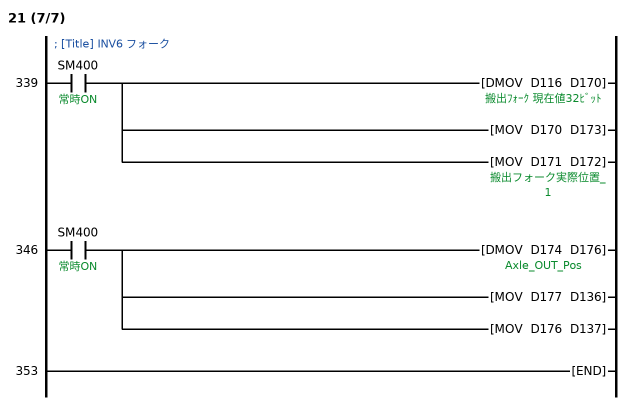
; [Title] INV6 フォーク
339   LD      SM400  ; 常時ON
      DMOV    D116 D170  ; 搬出ﾌｫｰｸ 現在値32ﾋﾞｯﾄ
      MOV     D170 D173
      MOV     D171 D172
346   LD      SM400  ; 常時ON
      DMOV    D174 D176
      MOV     D177 D136
      MOV     D176 D137
353   END
END_PROGRAM

PROGRAM 22  // Drive
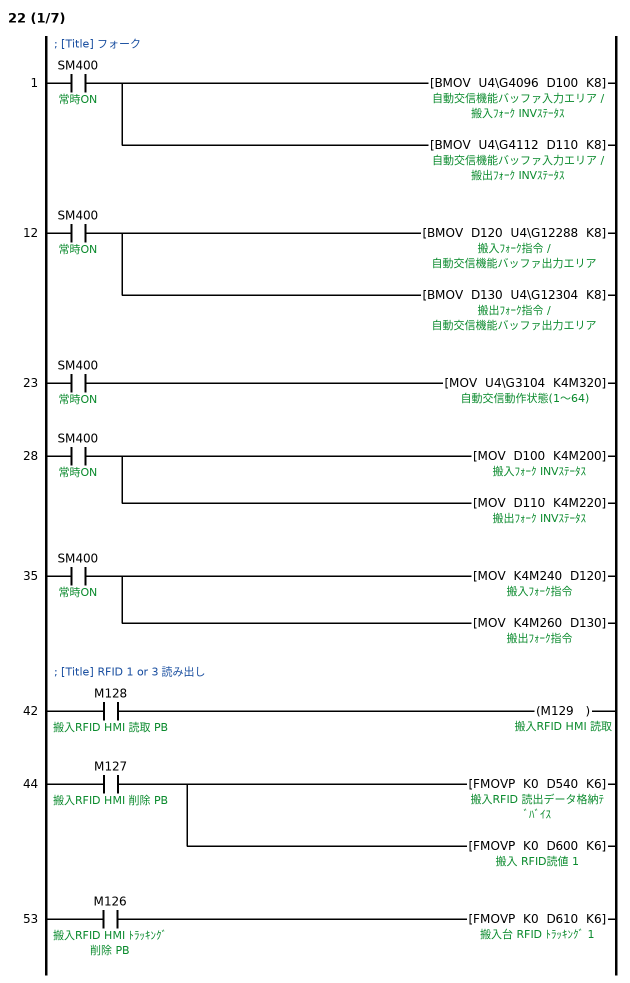
; [Title] フォーク
1     LD      SM400  ; 常時ON
      BMOV    U4\G4096 D100 K8  ; 自動交信機能バッファ入力エリア / 搬入ﾌｫｰｸ INVｽﾃｰﾀｽ
      BMOV    U4\G4112 D110 K8  ; 自動交信機能バッファ入力エリア / 搬出ﾌｫｰｸ INVｽﾃｰﾀｽ
12    LD      SM400  ; 常時ON
      BMOV    D120 U4\G12288 K8  ; 搬入ﾌｫｰｸ指令 / 自動交信機能バッファ出力エリア
      BMOV    D130 U4\G12304 K8  ; 搬出ﾌｫｰｸ指令 / 自動交信機能バッファ出力エリア
23    LD      SM400  ; 常時ON
      MOV     U4\G3104 K4M320  ; 自動交信動作状態(1～64) / INV2 通信異常
28    LD      SM400  ; 常時ON
      MOV     D100 K4M200  ; 搬入ﾌｫｰｸｽﾃｰﾀｽ 未使用
      MOV     D110 K4M220  ; 搬出ﾌｫｰｸｽﾃｰﾀｽ 未使用
35    LD      SM400  ; 常時ON
      MOV     K4M240 D120  ; 搬入ﾌｫｰｸ緊急停止
      MOV     K4M260 D130  ; 搬出ﾌｫｰｸ緊急停止
; [Title] RFID 1 or 3 読み出し
42    LD      M128  ; 搬入RFID HMI 読取 PB
      OUT     M129  ; 搬入RFID HMI 読取
44    LD      M127  ; 搬入RFID HMI 削除 PB
      FMOVP   K0 D540 K6  ; 搬入RFID 読出データ格納ﾃﾞﾊﾞｲｽ
      FMOVP   K0 D600 K6  ; 搬入 RFID読値 1
53    LD      M126  ; 搬入RFID HMI ﾄﾗｯｷﾝｸﾞ 削除 PB
      FMOVP   K0 D610 K6  ; 搬入台 RFID ﾄﾗｯｷﾝｸﾞ 1
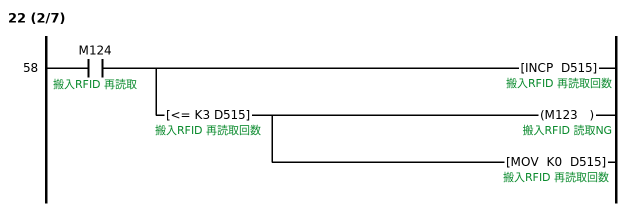
58    LD      M124  ; 搬入RFID 再読取
      INCP    D515  ; 搬入RFID 再読取回数
      AND<=   K3 D515  ; 搬入RFID 再読取回数
      OUT     M123  ; 搬入RFID 読取NG
      MOV     K0 D515
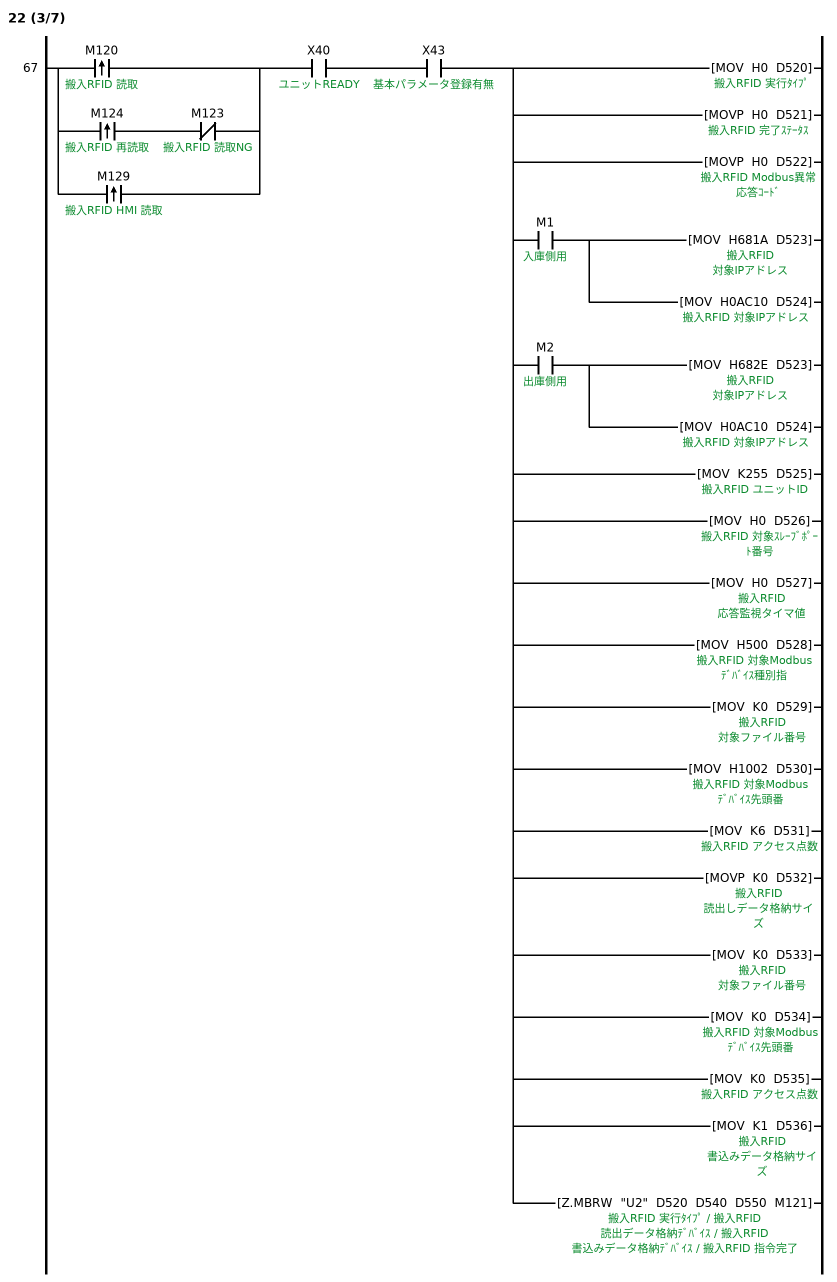
67    LDP     M120  ; 搬入RFID 読取
      LDP     M124  ; 搬入RFID 再読取
      ANI     M123  ; 搬入RFID 読取NG
      ORB
      ORP     M129  ; 搬入RFID HMI 読取
      AND     X40  ; ユニットREADY
      AND     X43  ; 基本パラメータ登録有無
      MOV     H0 D520  ; 搬入RFID 実行ﾀｲﾌﾟ
      MOVP    H0 D521  ; 搬入RFID 完了ｽﾃｰﾀｽ
      MOVP    H0 D522  ; 搬入RFID Modbus異常応答ｺｰﾄﾞ
      MPS
      AND     M1  ; 入庫側用
      MOV     H681A D523  ; 搬入RFID 対象IPアドレス
      MOV     H0AC10 D524  ; 搬入RFID 対象IPアドレス
      MRD
      AND     M2  ; 出庫側用
      MOV     H682E D523
      MOV     H0AC10 D524
      MPP
      MOV     K255 D525  ; 搬入RFID ユニットID
      MOV     H0 D526  ; 搬入RFID 対象ｽﾚｰﾌﾞﾎﾟｰﾄ番号
      MOV     H0 D527  ; 搬入RFID 応答監視タイマ値
      MOV     H500 D528  ; 搬入RFID 対象Modbusﾃﾞﾊﾞｲｽ種別指
      MOV     K0 D529  ; 搬入RFID 対象ファイル番号
      MOV     H1002 D530  ; 搬入RFID 対象Modbus ﾃﾞﾊﾞｲｽ先頭番
      MOV     K6 D531  ; 搬入RFID アクセス点数
      MOVP    K0 D532  ; 搬入RFID 読出しデータ格納サイズ
      MOV     K0 D533  ; 搬入RFID 対象ファイル番号
      MOV     K0 D534  ; 搬入RFID 対象Modbus ﾃﾞﾊﾞｲｽ先頭番
      MOV     K0 D535  ; 搬入RFID アクセス点数
      MOV     K1 D536  ; 搬入RFID 書込みデータ格納サイズ
      Z.MBRW  "U2" D520 D540 D550 M121  ; 搬入RFID 書込みデータ格納ﾃﾞﾊﾞｲｽ / 搬入RFID 指令完了
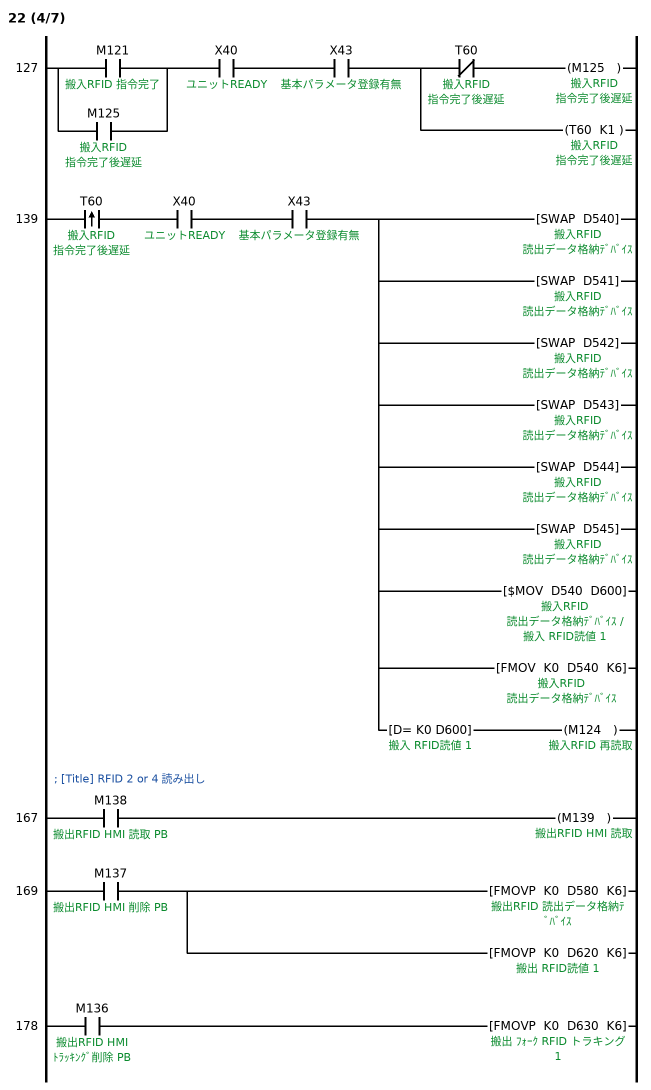
127   LD      M121  ; 搬入RFID 指令完了
      OR      M125  ; 搬入RFID 指令完了後遅延
      AND     X40  ; ユニットREADY
      AND     X43  ; 基本パラメータ登録有無
      MPS
      ANI     T60  ; 搬入RFID 指令完了後遅延
      OUT     M125  ; 搬入RFID 指令完了後遅延
      MPP
      OUT     T60 K1  ; 搬入RFID 指令完了後遅延
139   LDP     T60  ; 搬入RFID 指令完了後遅延
      AND     X40  ; ユニットREADY
      AND     X43  ; 基本パラメータ登録有無
      SWAP    D540
      SWAP    D541  ; 搬入RFID 読出データ格納ﾃﾞﾊﾞｲｽ
      SWAP    D542  ; 搬入RFID 読出データ格納ﾃﾞﾊﾞｲｽ
      SWAP    D543  ; 搬入RFID 読出データ格納ﾃﾞﾊﾞｲｽ
      SWAP    D544  ; 搬入RFID 読出データ格納ﾃﾞﾊﾞｲｽ
      SWAP    D545  ; 搬入RFID 読出データ格納ﾃﾞﾊﾞｲｽ
      $MOV    D540 D600
      FMOV    K0 D540 K6
      ANDD=   K0 D600  ; 搬入 RFID読値 1
      OUT     M124  ; 搬入RFID 再読取
; [Title] RFID 2 or 4 読み出し
167   LD      M138  ; 搬出RFID HMI 読取 PB
      OUT     M139  ; 搬出RFID HMI 読取
169   LD      M137  ; 搬出RFID HMI 削除 PB
      FMOVP   K0 D580 K6  ; 搬出RFID 読出データ格納ﾃﾞﾊﾞｲｽ
      FMOVP   K0 D620 K6  ; 搬出 RFID読値 1
178   LD      M136  ; 搬出RFID HMI ﾄﾗｯｷﾝｸﾞ削除 PB
      FMOVP   K0 D630 K6  ; 搬出 ﾌｫｰｸ RFID トラキング 1
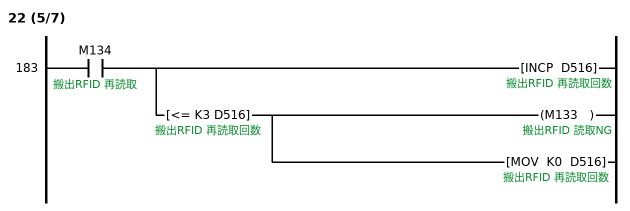
183   LD      M134  ; 搬出RFID 再読取
      INCP    D516  ; 搬出RFID 再読取回数
      AND<=   K3 D516  ; 搬出RFID 再読取回数
      OUT     M133  ; 搬出RFID 読取NG
      MOV     K0 D516
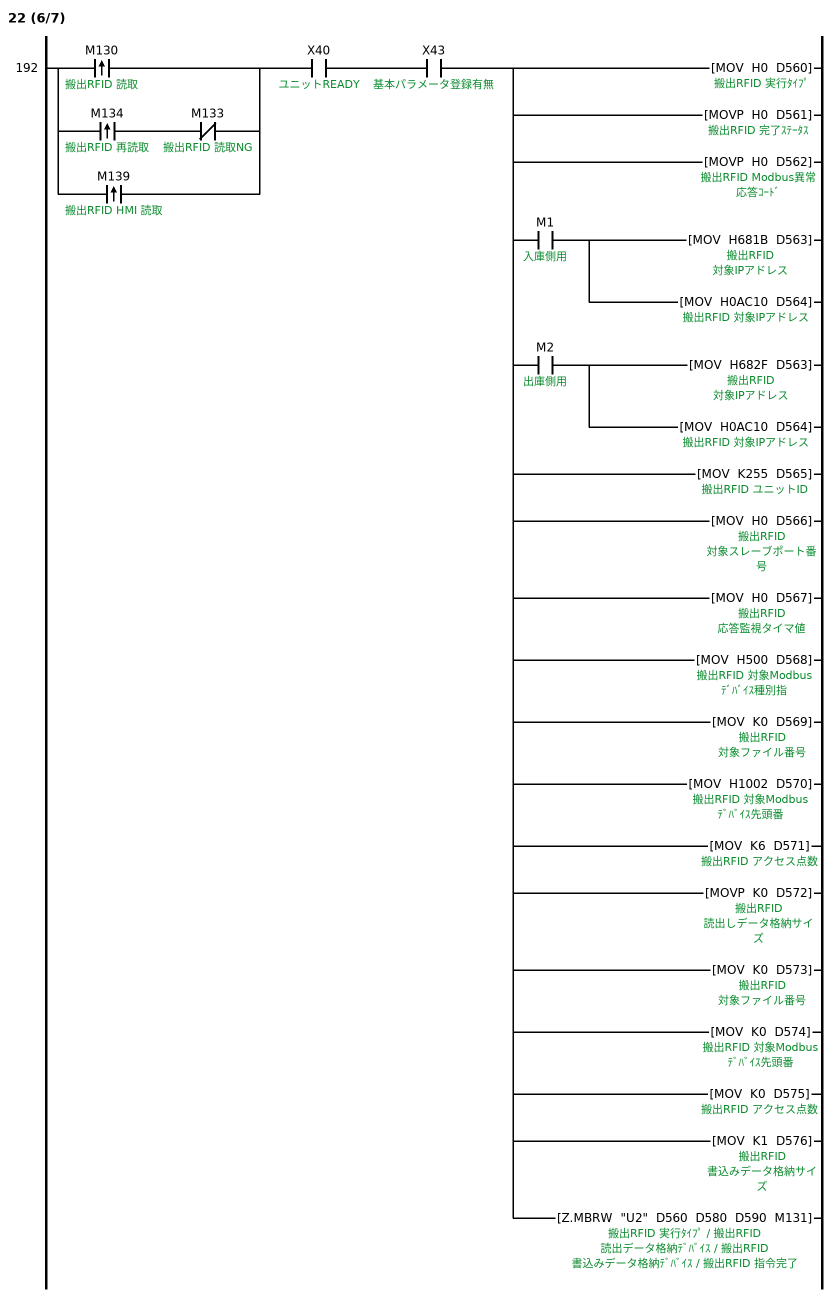
192   LDP     M130  ; 搬出RFID 読取
      LDP     M134  ; 搬出RFID 再読取
      ANI     M133  ; 搬出RFID 読取NG
      ORB
      ORP     M139  ; 搬出RFID HMI 読取
      AND     X40  ; ユニットREADY
      AND     X43  ; 基本パラメータ登録有無
      MOV     H0 D560  ; 搬出RFID 実行ﾀｲﾌﾟ
      MOVP    H0 D561  ; 搬出RFID 完了ｽﾃｰﾀｽ
      MOVP    H0 D562  ; 搬出RFID Modbus異常応答ｺｰﾄﾞ
      MPS
      AND     M1  ; 入庫側用
      MOV     H681B D563  ; 搬出RFID 対象IPアドレス
      MOV     H0AC10 D564  ; 搬出RFID 対象IPアドレス
      MRD
      AND     M2  ; 出庫側用
      MOV     H682F D563
      MOV     H0AC10 D564
      MPP
      MOV     K255 D565  ; 搬出RFID ユニットID
      MOV     H0 D566  ; 搬出RFID 対象スレーブポート番号
      MOV     H0 D567  ; 搬出RFID 応答監視タイマ値
      MOV     H500 D568  ; 搬出RFID 対象Modbusﾃﾞﾊﾞｲｽ種別指
      MOV     K0 D569  ; 搬出RFID 対象ファイル番号
      MOV     H1002 D570  ; 搬出RFID 対象Modbus ﾃﾞﾊﾞｲｽ先頭番
      MOV     K6 D571  ; 搬出RFID アクセス点数
      MOVP    K0 D572  ; 搬出RFID 読出しデータ格納サイズ
      MOV     K0 D573  ; 搬出RFID 対象ファイル番号
      MOV     K0 D574  ; 搬出RFID 対象Modbus ﾃﾞﾊﾞｲｽ先頭番
      MOV     K0 D575  ; 搬出RFID アクセス点数
      MOV     K1 D576  ; 搬出RFID 書込みデータ格納サイズ
      Z.MBRW  "U2" D560 D580 D590 M131  ; 搬出RFID 書込みデータ格納ﾃﾞﾊﾞｲｽ / 搬出RFID 指令完了
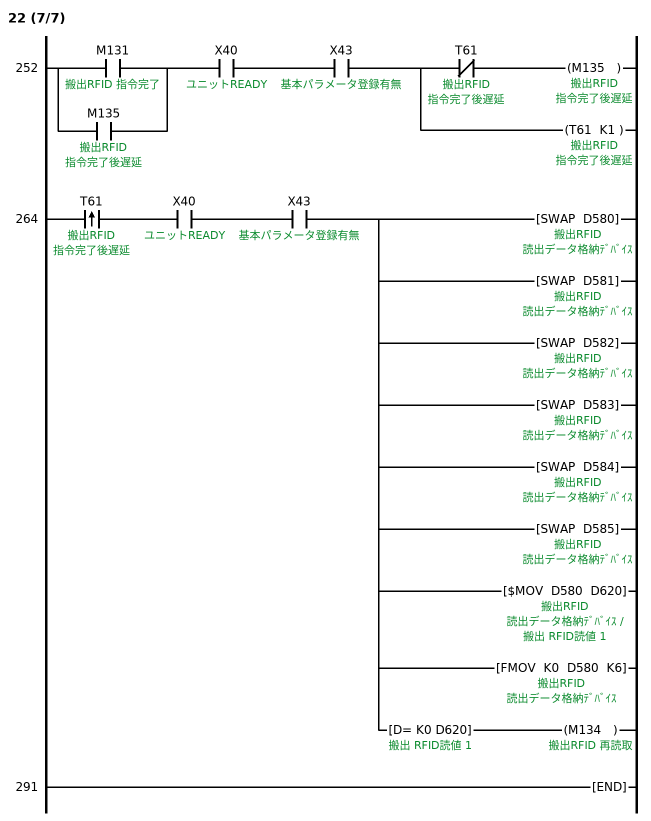
252   LD      M131  ; 搬出RFID 指令完了
      OR      M135  ; 搬出RFID 指令完了後遅延
      AND     X40  ; ユニットREADY
      AND     X43  ; 基本パラメータ登録有無
      MPS
      ANI     T61  ; 搬出RFID 指令完了後遅延
      OUT     M135  ; 搬出RFID 指令完了後遅延
      MPP
      OUT     T61 K1  ; 搬出RFID 指令完了後遅延
264   LDP     T61  ; 搬出RFID 指令完了後遅延
      AND     X40  ; ユニットREADY
      AND     X43  ; 基本パラメータ登録有無
      SWAP    D580
      SWAP    D581  ; 搬出RFID 読出データ格納ﾃﾞﾊﾞｲｽ
      SWAP    D582  ; 搬出RFID 読出データ格納ﾃﾞﾊﾞｲｽ
      SWAP    D583  ; 搬出RFID 読出データ格納ﾃﾞﾊﾞｲｽ
      SWAP    D584  ; 搬出RFID 読出データ格納ﾃﾞﾊﾞｲｽ
      SWAP    D585  ; 搬出RFID 読出データ格納ﾃﾞﾊﾞｲｽ
      $MOV    D580 D620
      FMOV    K0 D580 K6
      ANDD=   K0 D620  ; 搬出 RFID読値 1
      OUT     M134  ; 搬出RFID 再読取
291   END
END_PROGRAM

PROGRAM 30  // AGV
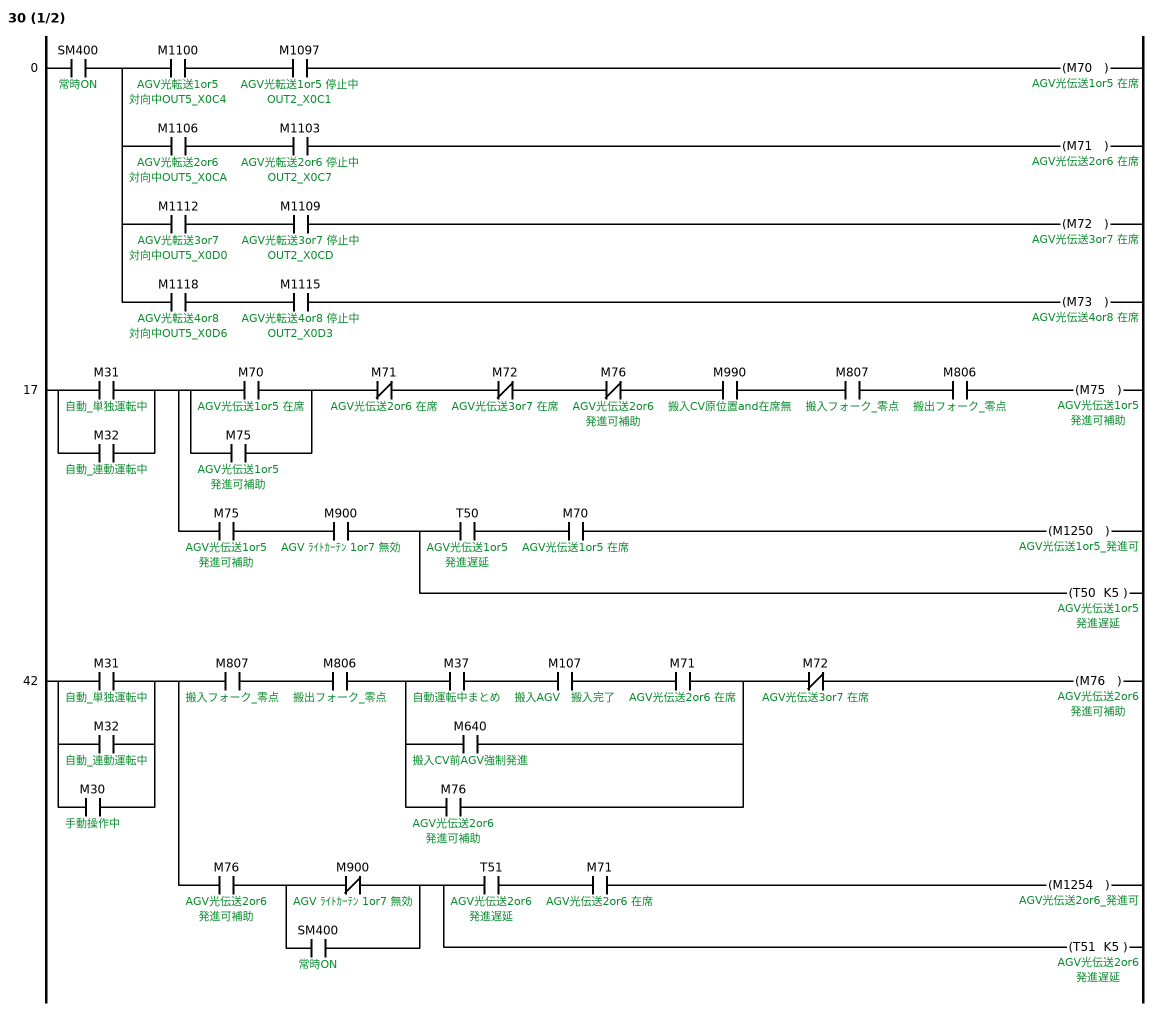
0     LD      SM400  ; 常時ON
      MPS
      AND     M1100  ; AGV光転送1or5 対向中OUT5_X0C4
      AND     M1097  ; AGV光転送1or5 停止中 OUT2_X0C1
      OUT     M70  ; AGV光伝送1or5 在席
      MRD
      AND     M1106  ; AGV光転送2or6 対向中OUT5_X0CA
      AND     M1103  ; AGV光転送2or6 停止中 OUT2_X0C7
      OUT     M71  ; AGV光伝送2or6 在席
      MRD
      AND     M1112  ; AGV光転送3or7 対向中OUT5_X0D0
      AND     M1109  ; AGV光転送3or7 停止中 OUT2_X0CD
      OUT     M72  ; AGV光伝送3or7 在席
      MPP
      AND     M1118  ; AGV光転送4or8 対向中OUT5_X0D6
      AND     M1115  ; AGV光転送4or8 停止中 OUT2_X0D3
      OUT     M73  ; AGV光伝送4or8 在席
17    LD      M31  ; 自動_単独運転中
      OR      M32  ; 自動_連動運転中
      MPS
      LD      M70  ; AGV光伝送1or5 在席
      OR      M75  ; AGV光伝送1or5 発進可補助
      ANB
      ANI     M71  ; AGV光伝送2or6 在席
      ANI     M72  ; AGV光伝送3or7 在席
      ANI     M76  ; AGV光伝送2or6 発進可補助
      AND     M990  ; 搬入CV原位置and在席無
      AND     M807  ; 搬入フォーク_零点
      AND     M806  ; 搬出フォーク_零点
      OUT     M75  ; AGV光伝送1or5 発進可補助
      MPP
      AND     M75  ; AGV光伝送1or5 発進可補助
      AND     M900  ; AGV ﾗｲﾄｶｰﾃﾝ 1or7 無効
      MPS
      AND     T50  ; AGV光伝送1or5 発進遅延
      AND     M70  ; AGV光伝送1or5 在席
      OUT     M1250  ; AGV光伝送1or5_発進可
      MPP
      OUT     T50 K5  ; AGV光伝送1or5 発進遅延
42    LD      M31  ; 自動_単独運転中
      OR      M32  ; 自動_連動運転中
      OR      M30  ; 手動操作中
      MPS
      AND     M807  ; 搬入フォーク_零点
      AND     M806  ; 搬出フォーク_零点
      LD      M37  ; 自動運転中まとめ
      AND     M107  ; 搬入AGV　搬入完了
      AND     M71  ; AGV光伝送2or6 在席
      OR      M640  ; 搬入CV前AGV強制発進
      OR      M76  ; AGV光伝送2or6 発進可補助
      ANB
      ANI     M72  ; AGV光伝送3or7 在席
      OUT     M76  ; AGV光伝送2or6 発進可補助
      MPP
      AND     M76  ; AGV光伝送2or6 発進可補助
      LDI     M900  ; AGV ﾗｲﾄｶｰﾃﾝ 1or7 無効
      OR      SM400  ; 常時ON
      ANB
      MPS
      AND     T51  ; AGV光伝送2or6 発進遅延
      AND     M71  ; AGV光伝送2or6 在席
      OUT     M1254  ; AGV光伝送2or6_発進可
      MPP
      OUT     T51 K5  ; AGV光伝送2or6 発進遅延
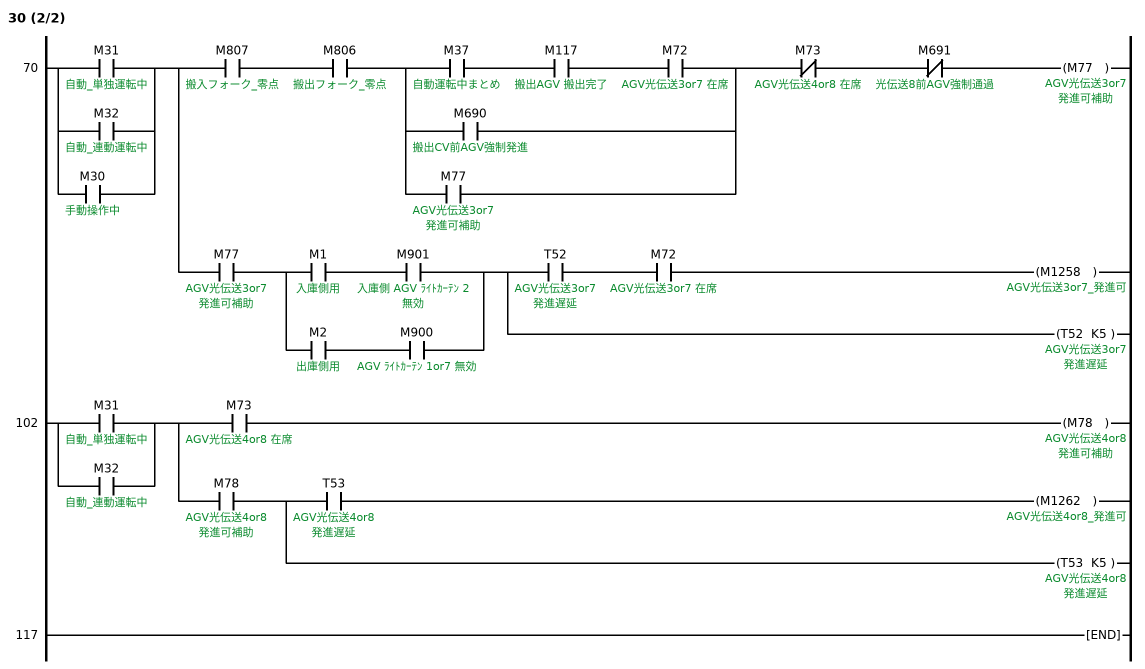
70    LD      M31  ; 自動_単独運転中
      OR      M32  ; 自動_連動運転中
      OR      M30  ; 手動操作中
      MPS
      AND     M807  ; 搬入フォーク_零点
      AND     M806  ; 搬出フォーク_零点
      LD      M37  ; 自動運転中まとめ
      AND     M117  ; 搬出AGV 搬出完了
      AND     M72  ; AGV光伝送3or7 在席
      OR      M690  ; 搬出CV前AGV強制発進
      OR      M77  ; AGV光伝送3or7 発進可補助
      ANB
      ANI     M73  ; AGV光伝送4or8 在席
      ANI     M691  ; 光伝送8前AGV強制通過
      OUT     M77  ; AGV光伝送3or7 発進可補助
      MPP
      AND     M77  ; AGV光伝送3or7 発進可補助
      LD      M1  ; 入庫側用
      AND     M901  ; 入庫側 AGV ﾗｲﾄｶｰﾃﾝ 2 無効
      LD      M2  ; 出庫側用
      AND     M900  ; AGV ﾗｲﾄｶｰﾃﾝ 1or7 無効
      ORB
      ANB
      MPS
      AND     T52  ; AGV光伝送3or7 発進遅延
      AND     M72  ; AGV光伝送3or7 在席
      OUT     M1258  ; AGV光伝送3or7_発進可
      MPP
      OUT     T52 K5  ; AGV光伝送3or7 発進遅延
102   LD      M31  ; 自動_単独運転中
      OR      M32  ; 自動_連動運転中
      MPS
      AND     M73  ; AGV光伝送4or8 在席
      OUT     M78  ; AGV光伝送4or8 発進可補助
      MPP
      AND     M78  ; AGV光伝送4or8 発進可補助
      MPS
      AND     T53  ; AGV光伝送4or8 発進遅延
      OUT     M1262  ; AGV光伝送4or8_発進可
      MPP
      OUT     T53 K5  ; AGV光伝送4or8 発進遅延
117   END
END_PROGRAM

PROGRAM 50  // IO 出力
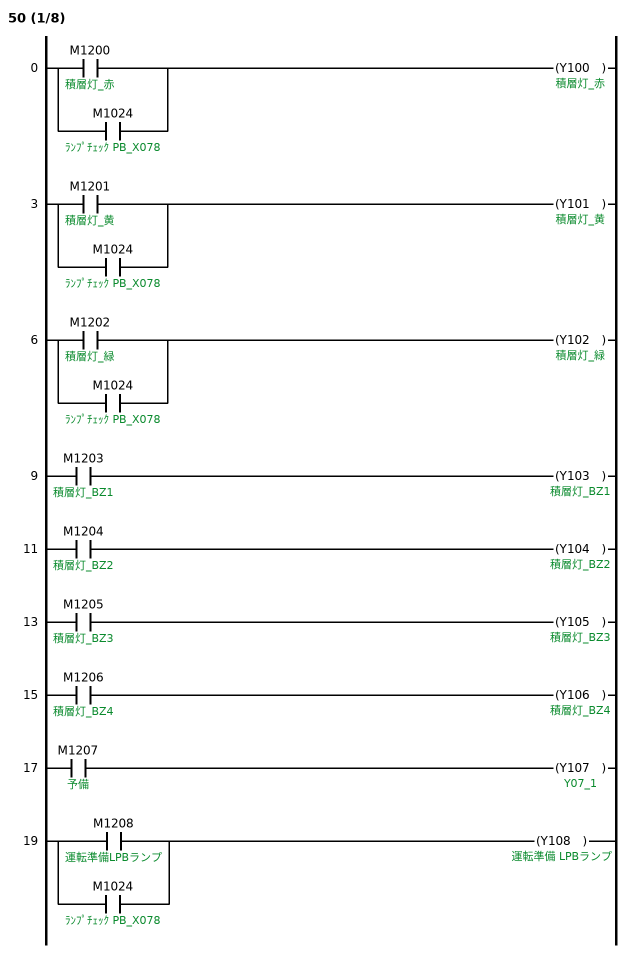
0     LD      M1200  ; 積層灯_赤
      OR      M1024  ; ﾗﾝﾌﾟﾁｪｯｸ PB_X078
      OUT     Y100  ; 積層灯_赤
3     LD      M1201  ; 積層灯_黄
      OR      M1024  ; ﾗﾝﾌﾟﾁｪｯｸ PB_X078
      OUT     Y101  ; 積層灯_黄
6     LD      M1202  ; 積層灯_緑
      OR      M1024  ; ﾗﾝﾌﾟﾁｪｯｸ PB_X078
      OUT     Y102  ; 積層灯_緑
9     LD      M1203  ; 積層灯_BZ1
      OUT     Y103  ; 積層灯_BZ1
11    LD      M1204  ; 積層灯_BZ2
      OUT     Y104  ; 積層灯_BZ2
13    LD      M1205  ; 積層灯_BZ3
      OUT     Y105  ; 積層灯_BZ3
15    LD      M1206  ; 積層灯_BZ4
      OUT     Y106  ; 積層灯_BZ4
17    LD      M1207  ; 予備
      OUT     Y107  ; Y07_1
19    LD      M1208  ; 運転準備LPBランプ
      OR      M1024  ; ﾗﾝﾌﾟﾁｪｯｸ PB_X078
      OUT     Y108  ; 運転準備 LPBランプ
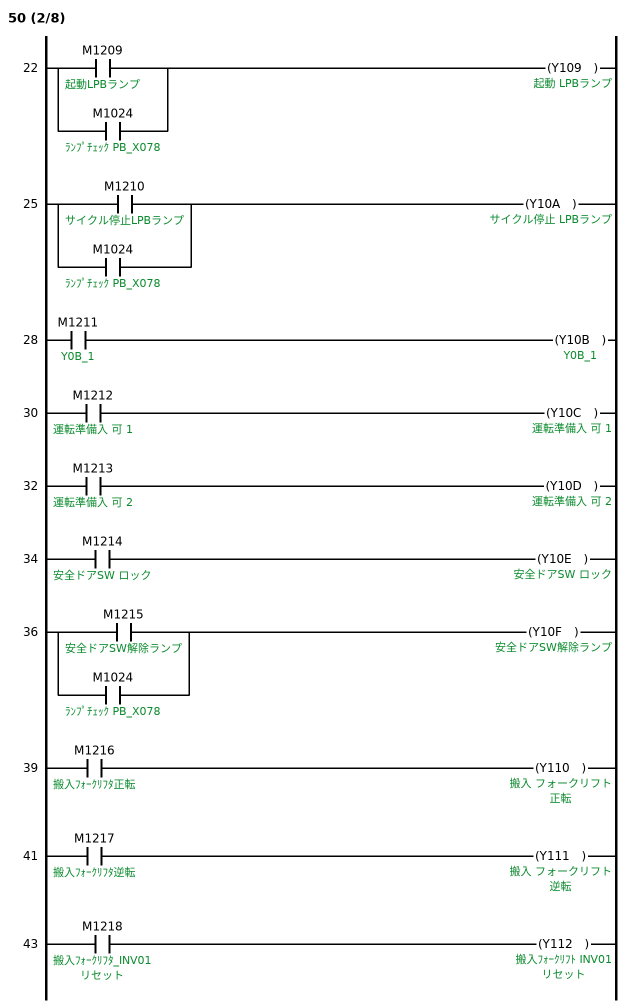
22    LD      M1209  ; 起動LPBランプ
      OR      M1024  ; ﾗﾝﾌﾟﾁｪｯｸ PB_X078
      OUT     Y109  ; 起動 LPBランプ
25    LD      M1210  ; サイクル停止LPBランプ
      OR      M1024  ; ﾗﾝﾌﾟﾁｪｯｸ PB_X078
      OUT     Y10A  ; サイクル停止 LPBランプ
28    LD      M1211  ; Y0B_1
      OUT     Y10B  ; Y0B_1
30    LD      M1212  ; 運転準備入 可 1
      OUT     Y10C  ; 運転準備入 可 1
32    LD      M1213  ; 運転準備入 可 2
      OUT     Y10D  ; 運転準備入 可 2
34    LD      M1214  ; 安全ドアSW ロック
      OUT     Y10E  ; 安全ドアSW ロック
36    LD      M1215  ; 安全ドアSW解除ランプ
      OR      M1024  ; ﾗﾝﾌﾟﾁｪｯｸ PB_X078
      OUT     Y10F  ; 安全ドアSW解除ランプ
39    LD      M1216  ; 搬入ﾌｫｰｸﾘﾌﾀ正転
      OUT     Y110  ; 搬入 フォークリフト 正転
41    LD      M1217  ; 搬入ﾌｫｰｸﾘﾌﾀ逆転
      OUT     Y111  ; 搬入 フォークリフト 逆転
43    LD      M1218  ; 搬入ﾌｫｰｸﾘﾌﾀ_INV01 リセット
      OUT     Y112  ; 搬入ﾌｫｰｸﾘﾌﾄ INV01 リセット
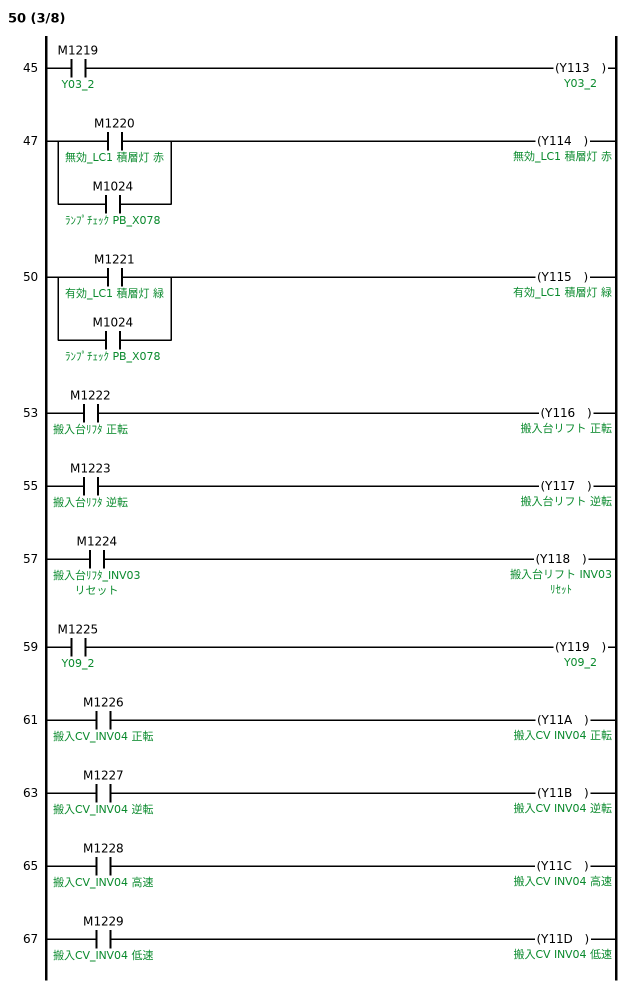
45    LD      M1219  ; Y03_2
      OUT     Y113  ; Y03_2
47    LD      M1220  ; 無効_LC1 積層灯 赤
      OR      M1024  ; ﾗﾝﾌﾟﾁｪｯｸ PB_X078
      OUT     Y114  ; 無効_LC1 積層灯 赤
50    LD      M1221  ; 有効_LC1 積層灯 緑
      OR      M1024  ; ﾗﾝﾌﾟﾁｪｯｸ PB_X078
      OUT     Y115  ; 有効_LC1 積層灯 緑
53    LD      M1222  ; 搬入台ﾘﾌﾀ 正転
      OUT     Y116  ; 搬入台リフト 正転
55    LD      M1223  ; 搬入台ﾘﾌﾀ 逆転
      OUT     Y117  ; 搬入台リフト 逆転
57    LD      M1224  ; 搬入台ﾘﾌﾀ_INV03 リセット
      OUT     Y118  ; 搬入台リフト INV03 ﾘｾｯﾄ
59    LD      M1225  ; Y09_2
      OUT     Y119  ; Y09_2
61    LD      M1226  ; 搬入CV_INV04 正転
      OUT     Y11A  ; 搬入CV INV04 正転
63    LD      M1227  ; 搬入CV_INV04 逆転
      OUT     Y11B  ; 搬入CV INV04 逆転
65    LD      M1228  ; 搬入CV_INV04 高速
      OUT     Y11C  ; 搬入CV INV04 高速
67    LD      M1229  ; 搬入CV_INV04 低速
      OUT     Y11D  ; 搬入CV INV04 低速
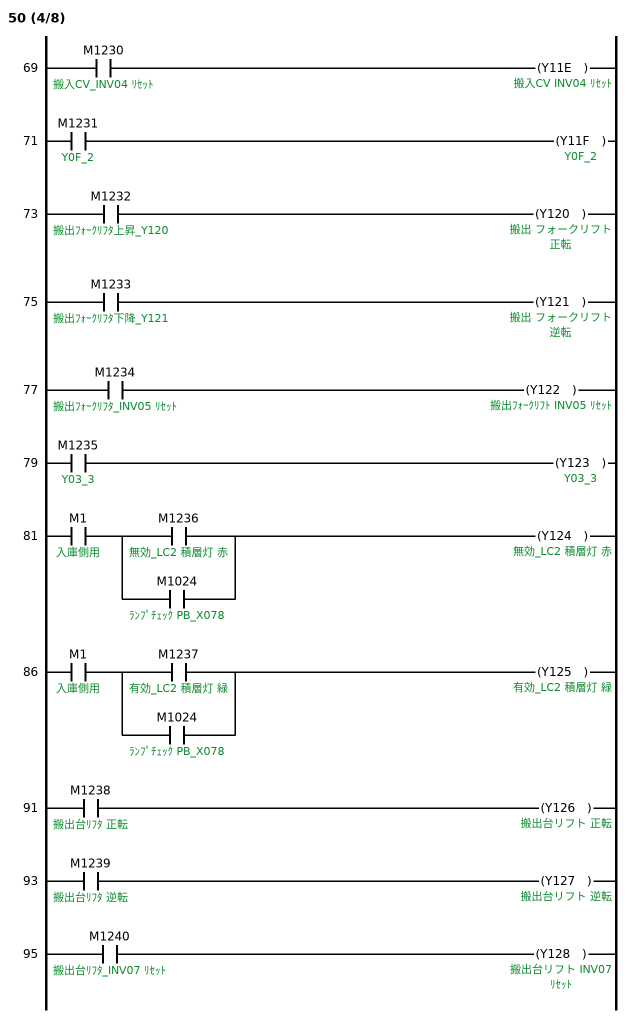
69    LD      M1230  ; 搬入CV_INV04 ﾘｾｯﾄ
      OUT     Y11E  ; 搬入CV INV04 ﾘｾｯﾄ
71    LD      M1231  ; Y0F_2
      OUT     Y11F  ; Y0F_2
73    LD      M1232  ; 搬出ﾌｫｰｸﾘﾌﾀ上昇_Y120
      OUT     Y120  ; 搬出 フォークリフト 正転
75    LD      M1233  ; 搬出ﾌｫｰｸﾘﾌﾀ下降_Y121
      OUT     Y121  ; 搬出 フォークリフト 逆転
77    LD      M1234  ; 搬出ﾌｫｰｸﾘﾌﾀ_INV05 ﾘｾｯﾄ
      OUT     Y122  ; 搬出ﾌｫｰｸﾘﾌﾄ INV05 ﾘｾｯﾄ
79    LD      M1235  ; Y03_3
      OUT     Y123  ; Y03_3
81    LD      M1  ; 入庫側用
      LD      M1236  ; 無効_LC2 積層灯 赤
      OR      M1024  ; ﾗﾝﾌﾟﾁｪｯｸ PB_X078
      ANB
      OUT     Y124  ; 無効_LC2 積層灯 赤
86    LD      M1  ; 入庫側用
      LD      M1237  ; 有効_LC2 積層灯 緑
      OR      M1024  ; ﾗﾝﾌﾟﾁｪｯｸ PB_X078
      ANB
      OUT     Y125  ; 有効_LC2 積層灯 緑
91    LD      M1238  ; 搬出台ﾘﾌﾀ 正転
      OUT     Y126  ; 搬出台リフト 正転
93    LD      M1239  ; 搬出台ﾘﾌﾀ 逆転
      OUT     Y127  ; 搬出台リフト 逆転
95    LD      M1240  ; 搬出台ﾘﾌﾀ_INV07 ﾘｾｯﾄ
      OUT     Y128  ; 搬出台リフト INV07 ﾘｾｯﾄ
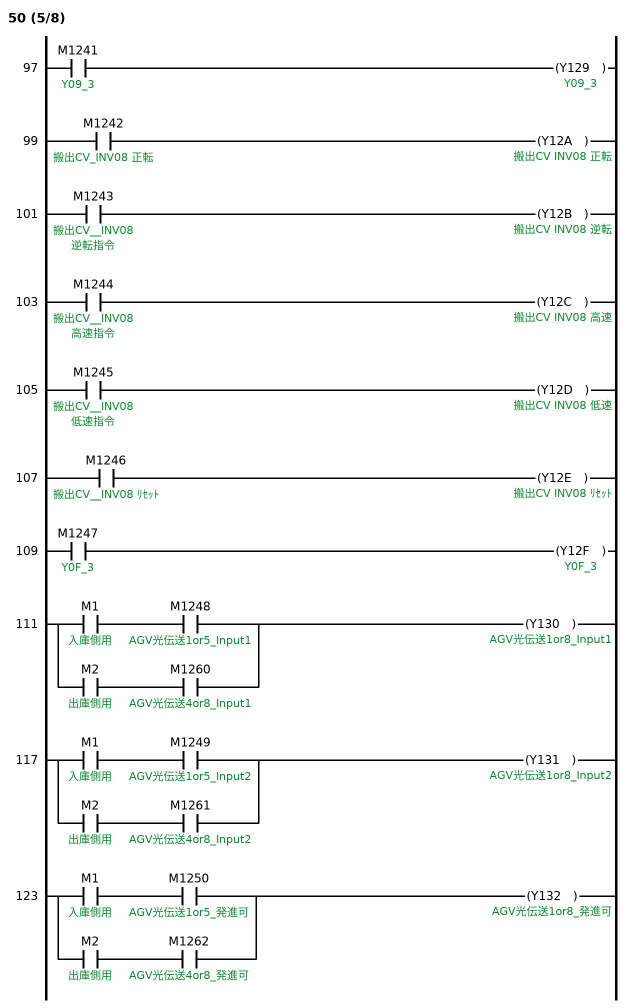
97    LD      M1241  ; Y09_3
      OUT     Y129  ; Y09_3
99    LD      M1242  ; 搬出CV_INV08 正転
      OUT     Y12A  ; 搬出CV INV08 正転
101   LD      M1243  ; 搬出CV__INV08 逆転指令
      OUT     Y12B  ; 搬出CV INV08 逆転
103   LD      M1244  ; 搬出CV__INV08 高速指令
      OUT     Y12C  ; 搬出CV INV08 高速
105   LD      M1245  ; 搬出CV__INV08 低速指令
      OUT     Y12D  ; 搬出CV INV08 低速
107   LD      M1246  ; 搬出CV__INV08 ﾘｾｯﾄ
      OUT     Y12E  ; 搬出CV INV08 ﾘｾｯﾄ
109   LD      M1247  ; Y0F_3
      OUT     Y12F  ; Y0F_3
111   LD      M1  ; 入庫側用
      AND     M1248  ; AGV光伝送1or5_Input1
      LD      M2  ; 出庫側用
      AND     M1260  ; AGV光伝送4or8_Input1
      ORB
      OUT     Y130  ; AGV光伝送1or8_Input1
117   LD      M1  ; 入庫側用
      AND     M1249  ; AGV光伝送1or5_Input2
      LD      M2  ; 出庫側用
      AND     M1261  ; AGV光伝送4or8_Input2
      ORB
      OUT     Y131  ; AGV光伝送1or8_Input2
123   LD      M1  ; 入庫側用
      AND     M1250  ; AGV光伝送1or5_発進可
      LD      M2  ; 出庫側用
      AND     M1262  ; AGV光伝送4or8_発進可
      ORB
      OUT     Y132  ; AGV光伝送1or8_発進可
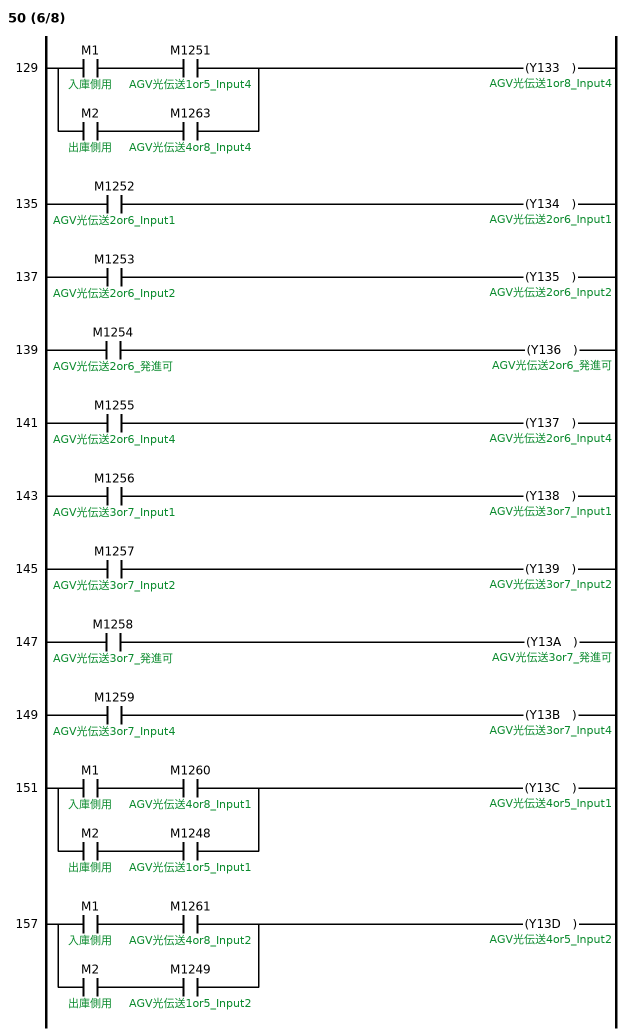
129   LD      M1  ; 入庫側用
      AND     M1251  ; AGV光伝送1or5_Input4
      LD      M2  ; 出庫側用
      AND     M1263  ; AGV光伝送4or8_Input4
      ORB
      OUT     Y133  ; AGV光伝送1or8_Input4
135   LD      M1252  ; AGV光伝送2or6_Input1
      OUT     Y134  ; AGV光伝送2or6_Input1
137   LD      M1253  ; AGV光伝送2or6_Input2
      OUT     Y135  ; AGV光伝送2or6_Input2
139   LD      M1254  ; AGV光伝送2or6_発進可
      OUT     Y136  ; AGV光伝送2or6_発進可
141   LD      M1255  ; AGV光伝送2or6_Input4
      OUT     Y137  ; AGV光伝送2or6_Input4
143   LD      M1256  ; AGV光伝送3or7_Input1
      OUT     Y138  ; AGV光伝送3or7_Input1
145   LD      M1257  ; AGV光伝送3or7_Input2
      OUT     Y139  ; AGV光伝送3or7_Input2
147   LD      M1258  ; AGV光伝送3or7_発進可
      OUT     Y13A  ; AGV光伝送3or7_発進可
149   LD      M1259  ; AGV光伝送3or7_Input4
      OUT     Y13B  ; AGV光伝送3or7_Input4
151   LD      M1  ; 入庫側用
      AND     M1260  ; AGV光伝送4or8_Input1
      LD      M2  ; 出庫側用
      AND     M1248  ; AGV光伝送1or5_Input1
      ORB
      OUT     Y13C  ; AGV光伝送4or5_Input1
157   LD      M1  ; 入庫側用
      AND     M1261  ; AGV光伝送4or8_Input2
      LD      M2  ; 出庫側用
      AND     M1249  ; AGV光伝送1or5_Input2
      ORB
      OUT     Y13D  ; AGV光伝送4or5_Input2
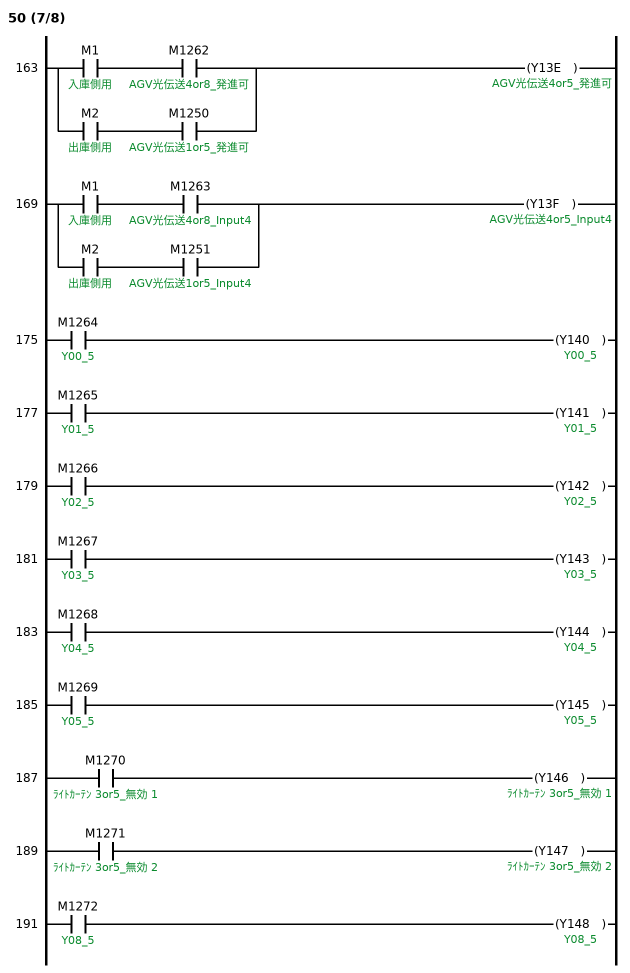
163   LD      M1  ; 入庫側用
      AND     M1262  ; AGV光伝送4or8_発進可
      LD      M2  ; 出庫側用
      AND     M1250  ; AGV光伝送1or5_発進可
      ORB
      OUT     Y13E  ; AGV光伝送4or5_発進可
169   LD      M1  ; 入庫側用
      AND     M1263  ; AGV光伝送4or8_Input4
      LD      M2  ; 出庫側用
      AND     M1251  ; AGV光伝送1or5_Input4
      ORB
      OUT     Y13F  ; AGV光伝送4or5_Input4
175   LD      M1264  ; Y00_5
      OUT     Y140  ; Y00_5
177   LD      M1265  ; Y01_5
      OUT     Y141  ; Y01_5
179   LD      M1266  ; Y02_5
      OUT     Y142  ; Y02_5
181   LD      M1267  ; Y03_5
      OUT     Y143  ; Y03_5
183   LD      M1268  ; Y04_5
      OUT     Y144  ; Y04_5
185   LD      M1269  ; Y05_5
      OUT     Y145  ; Y05_5
187   LD      M1270  ; ﾗｲﾄｶｰﾃﾝ 3or5_無効 1
      OUT     Y146  ; ﾗｲﾄｶｰﾃﾝ 3or5_無効 1
189   LD      M1271  ; ﾗｲﾄｶｰﾃﾝ 3or5_無効 2
      OUT     Y147  ; ﾗｲﾄｶｰﾃﾝ 3or5_無効 2
191   LD      M1272  ; Y08_5
      OUT     Y148  ; Y08_5
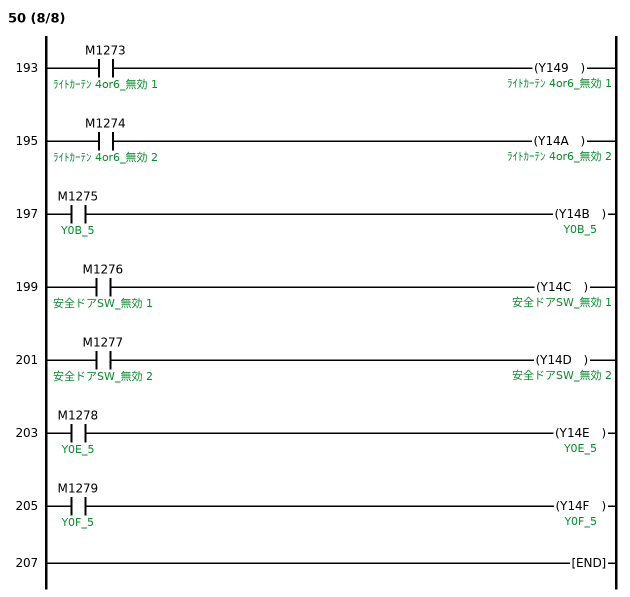
193   LD      M1273  ; ﾗｲﾄｶｰﾃﾝ 4or6_無効 1
      OUT     Y149  ; ﾗｲﾄｶｰﾃﾝ 4or6_無効 1
195   LD      M1274  ; ﾗｲﾄｶｰﾃﾝ 4or6_無効 2
      OUT     Y14A  ; ﾗｲﾄｶｰﾃﾝ 4or6_無効 2
197   LD      M1275  ; Y0B_5
      OUT     Y14B  ; Y0B_5
199   LD      M1276  ; 安全ドアSW_無効 1
      OUT     Y14C  ; 安全ドアSW_無効 1
201   LD      M1277  ; 安全ドアSW_無効 2
      OUT     Y14D  ; 安全ドアSW_無効 2
203   LD      M1278  ; Y0E_5
      OUT     Y14E  ; Y0E_5
205   LD      M1279  ; Y0F_5
      OUT     Y14F  ; Y0F_5
207   END
END_PROGRAM

PROGRAM 51A  // CC-LinkIE XVD 出力
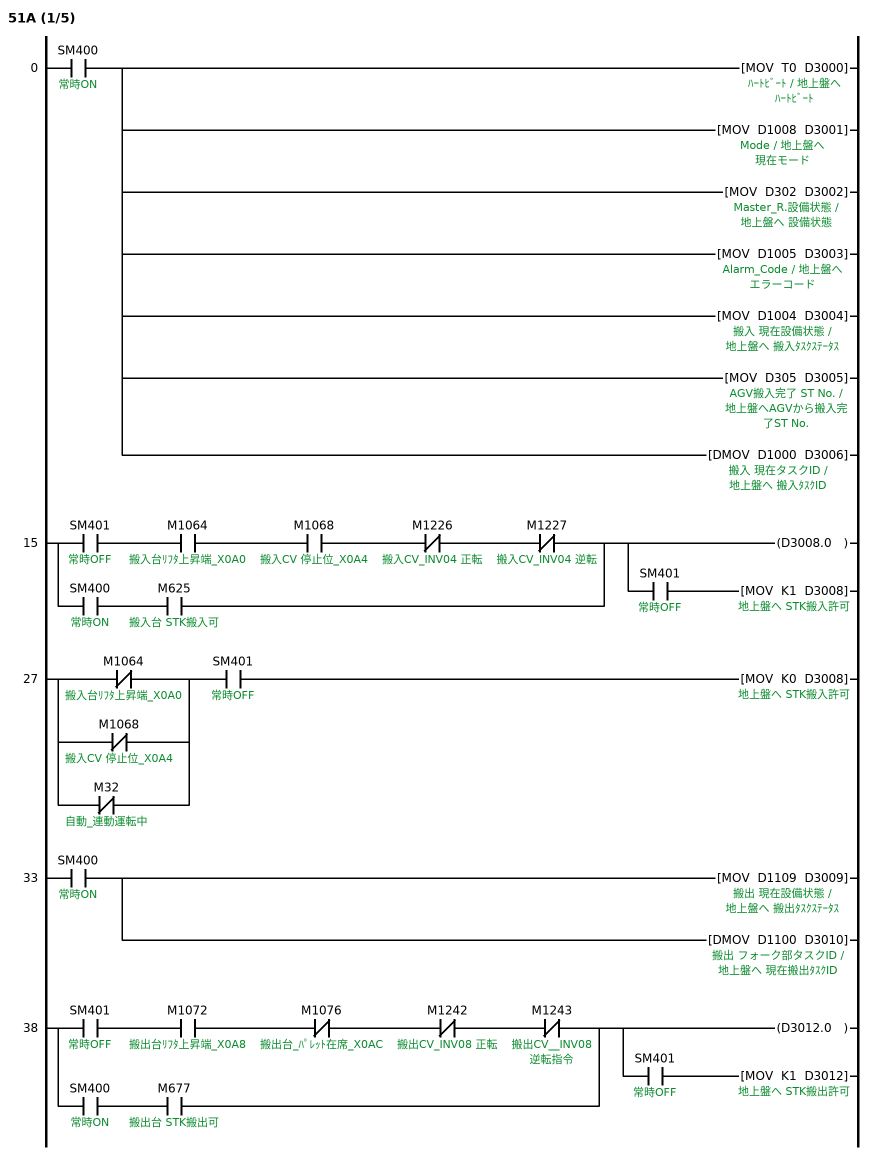
0     LD      SM400  ; 常時ON
      MOV     T0 D3000  ; ﾊｰﾄﾋﾞｰﾄ / 地上盤へ ﾊｰﾄﾋﾞｰﾄ
      MOV     D1008 D3001  ; Mode / 地上盤へ 現在モード
      MOV     D302 D3002  ; Master_R.設備状態 / 地上盤へ 設備状態
      MOV     D1005 D3003  ; Alarm_Code / 地上盤へ エラーコード
      MOV     D1004 D3004  ; 搬入 現在設備状態 / 地上盤へ 搬入ﾀｽｸｽﾃｰﾀｽ
      MOV     D305 D3005  ; AGV搬入完了 ST No. / 地上盤へAGVから搬入完了ST No.
      DMOV    D1000 D3006  ; 搬入 現在タスクID / 地上盤へ 搬入ﾀｽｸID
15    LD      SM401  ; 常時OFF
      AND     M1064  ; 搬入台ﾘﾌﾀ上昇端_X0A0
      AND     M1068  ; 搬入CV 停止位_X0A4
      ANI     M1226  ; 搬入CV_INV04 正転
      ANI     M1227  ; 搬入CV_INV04 逆転
      LD      SM400  ; 常時ON
      AND     M625  ; 搬入台 STK搬入可
      ORB
      OUT     D3008.0
      AND     SM401  ; 常時OFF
      MOV     K1 D3008  ; 地上盤へ STK搬入許可
27    LDI     M1064  ; 搬入台ﾘﾌﾀ上昇端_X0A0
      ORI     M1068  ; 搬入CV 停止位_X0A4
      ORI     M32  ; 自動_連動運転中
      AND     SM401  ; 常時OFF
      MOV     K0 D3008
33    LD      SM400  ; 常時ON
      MOV     D1109 D3009  ; 搬出 現在設備状態 / 地上盤へ 搬出ﾀｽｸｽﾃｰﾀｽ
      DMOV    D1100 D3010  ; 搬出 フォーク部タスクID / 地上盤へ 現在搬出ﾀｽｸID
38    LD      SM401  ; 常時OFF
      AND     M1072  ; 搬出台ﾘﾌﾀ上昇端_X0A8
      ANI     M1076  ; 搬出台_ﾊﾟﾚｯﾄ在席_X0AC
      ANI     M1242  ; 搬出CV_INV08 正転
      ANI     M1243  ; 搬出CV__INV08 逆転指令
      LD      SM400  ; 常時ON
      AND     M677  ; 搬出台 STK搬出可
      ORB
      OUT     D3012.0
      AND     SM401  ; 常時OFF
      MOV     K1 D3012  ; 地上盤へ STK搬出許可
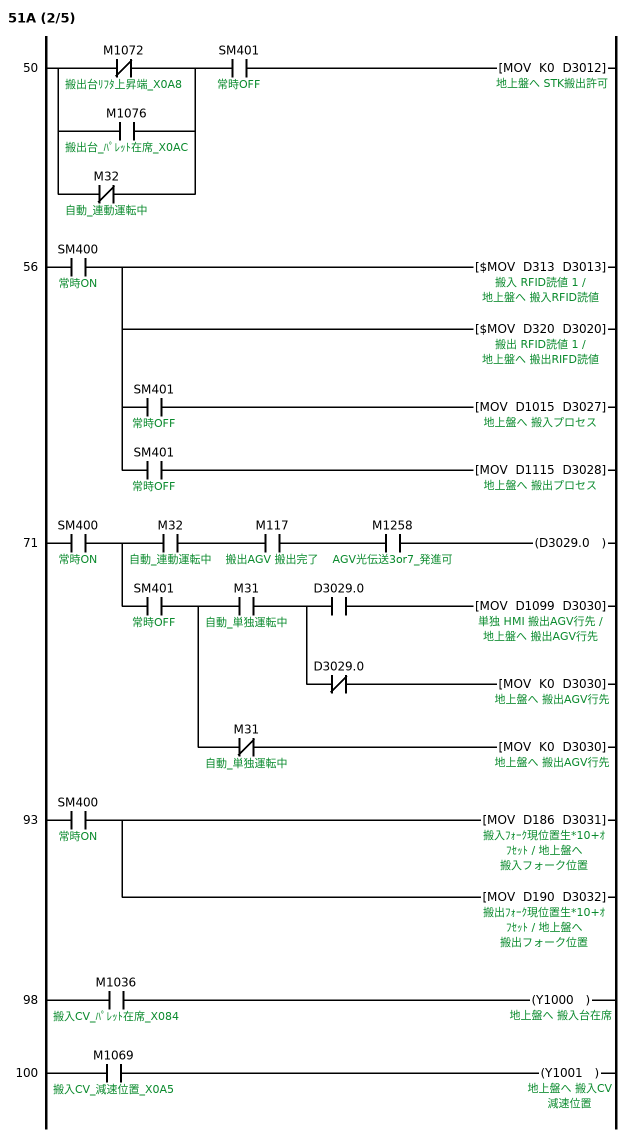
50    LDI     M1072  ; 搬出台ﾘﾌﾀ上昇端_X0A8
      OR      M1076  ; 搬出台_ﾊﾟﾚｯﾄ在席_X0AC
      ORI     M32  ; 自動_連動運転中
      AND     SM401  ; 常時OFF
      MOV     K0 D3012
56    LD      SM400  ; 常時ON
      $MOV    D313 D3013  ; 搬入 RFID読値 1 / 地上盤へ 搬入RFID読値
      $MOV    D320 D3020  ; 搬出 RFID読値 1 / 地上盤へ 搬出RIFD読値
      MPS
      AND     SM401  ; 常時OFF
      MOV     D1015 D3027  ; 地上盤へ 搬入プロセス
      MPP
      AND     SM401  ; 常時OFF
      MOV     D1115 D3028  ; 地上盤へ 搬出プロセス
71    LD      SM400  ; 常時ON
      MPS
      AND     M32  ; 自動_連動運転中
      AND     M117  ; 搬出AGV 搬出完了
      AND     M1258  ; AGV光伝送3or7_発進可
      OUT     D3029.0
      MPP
      AND     SM401  ; 常時OFF
      MPS
      AND     M31  ; 自動_単独運転中
      MPS
      AND     D3029.0
      MOV     D1099 D3030  ; 単独 HMI 搬出AGV行先 / 地上盤へ 搬出AGV行先
      MPP
      ANI     D3029.0
      MOV     K0 D3030
      MPP
      ANI     M31  ; 自動_単独運転中
      MOV     K0 D3030
93    LD      SM400  ; 常時ON
      MOV     D186 D3031  ; 搬入ﾌｫｰｸ現位置生*10+ｵﾌｾｯﾄ / 地上盤へ 搬入フォーク位置
      MOV     D190 D3032  ; 搬出ﾌｫｰｸ現位置生*10+ｵﾌｾｯﾄ / 地上盤へ 搬出フォーク位置
98    LD      M1036  ; 搬入CV_ﾊﾟﾚｯﾄ在席_X084
      OUT     Y1000  ; 地上盤へ 搬入台在席
100   LD      M1069  ; 搬入CV_減速位置_X0A5
      OUT     Y1001  ; 地上盤へ 搬入CV 減速位置
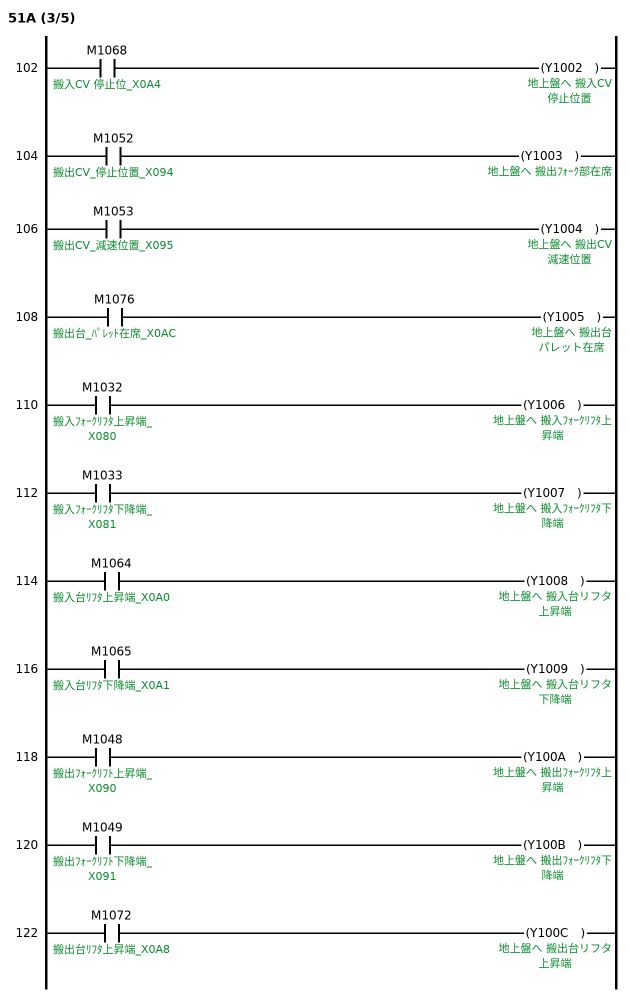
102   LD      M1068  ; 搬入CV 停止位_X0A4
      OUT     Y1002  ; 地上盤へ 搬入CV 停止位置
104   LD      M1052  ; 搬出CV_停止位置_X094
      OUT     Y1003  ; 地上盤へ 搬出ﾌｫｰｸ部在席
106   LD      M1053  ; 搬出CV_減速位置_X095
      OUT     Y1004  ; 地上盤へ 搬出CV 減速位置
108   LD      M1076  ; 搬出台_ﾊﾟﾚｯﾄ在席_X0AC
      OUT     Y1005  ; 地上盤へ 搬出台 パレット在席
110   LD      M1032  ; 搬入ﾌｫｰｸﾘﾌﾀ上昇端_X080
      OUT     Y1006  ; 地上盤へ 搬入ﾌｫｰｸﾘﾌﾀ上昇端
112   LD      M1033  ; 搬入ﾌｫｰｸﾘﾌﾀ下降端_X081
      OUT     Y1007  ; 地上盤へ 搬入ﾌｫｰｸﾘﾌﾀ下降端
114   LD      M1064  ; 搬入台ﾘﾌﾀ上昇端_X0A0
      OUT     Y1008  ; 地上盤へ 搬入台リフタ 上昇端
116   LD      M1065  ; 搬入台ﾘﾌﾀ下降端_X0A1
      OUT     Y1009  ; 地上盤へ 搬入台リフタ 下降端
118   LD      M1048  ; 搬出ﾌｫｰｸﾘﾌﾄ上昇端_X090
      OUT     Y100A  ; 地上盤へ 搬出ﾌｫｰｸﾘﾌﾀ上昇端
120   LD      M1049  ; 搬出ﾌｫｰｸﾘﾌﾄ下降端_X091
      OUT     Y100B  ; 地上盤へ 搬出ﾌｫｰｸﾘﾌﾀ下降端
122   LD      M1072  ; 搬出台ﾘﾌﾀ上昇端_X0A8
      OUT     Y100C  ; 地上盤へ 搬出台リフタ 上昇端
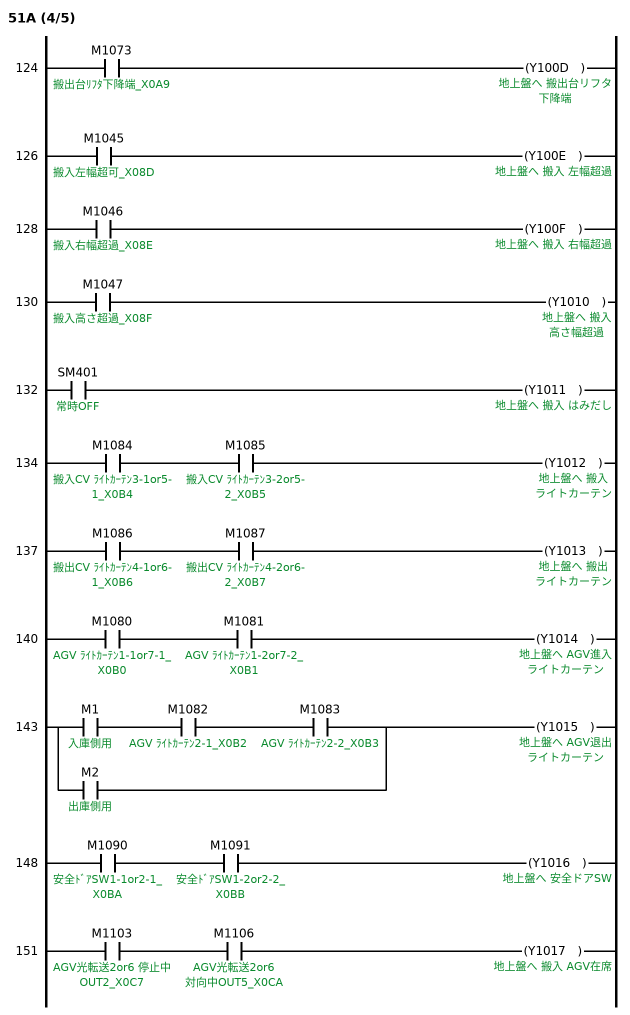
124   LD      M1073  ; 搬出台ﾘﾌﾀ下降端_X0A9
      OUT     Y100D  ; 地上盤へ 搬出台リフタ 下降端
126   LD      M1045  ; 搬入左幅超可_X08D
      OUT     Y100E  ; 地上盤へ 搬入 左幅超過
128   LD      M1046  ; 搬入右幅超過_X08E
      OUT     Y100F  ; 地上盤へ 搬入 右幅超過
130   LD      M1047  ; 搬入高さ超過_X08F
      OUT     Y1010  ; 地上盤へ 搬入 高さ幅超過
132   LD      SM401  ; 常時OFF
      OUT     Y1011  ; 地上盤へ 搬入 はみだし
134   LD      M1084  ; 搬入CV ﾗｲﾄｶｰﾃﾝ3-1or5-1_X0B4
      AND     M1085  ; 搬入CV ﾗｲﾄｶｰﾃﾝ3-2or5-2_X0B5
      OUT     Y1012  ; 地上盤へ 搬入 ライトカーテン
137   LD      M1086  ; 搬出CV ﾗｲﾄｶｰﾃﾝ4-1or6-1_X0B6
      AND     M1087  ; 搬出CV ﾗｲﾄｶｰﾃﾝ4-2or6-2_X0B7
      OUT     Y1013  ; 地上盤へ 搬出 ライトカーテン
140   LD      M1080  ; AGV ﾗｲﾄｶｰﾃﾝ1-1or7-1_X0B0
      AND     M1081  ; AGV ﾗｲﾄｶｰﾃﾝ1-2or7-2_X0B1
      OUT     Y1014  ; 地上盤へ AGV進入 ライトカーテン
143   LD      M1  ; 入庫側用
      AND     M1082  ; AGV ﾗｲﾄｶｰﾃﾝ2-1_X0B2
      AND     M1083  ; AGV ﾗｲﾄｶｰﾃﾝ2-2_X0B3
      OR      M2  ; 出庫側用
      OUT     Y1015  ; 地上盤へ AGV退出 ライトカーテン
148   LD      M1090  ; 安全ﾄﾞｱSW1-1or2-1_X0BA
      AND     M1091  ; 安全ﾄﾞｱSW1-2or2-2_X0BB
      OUT     Y1016  ; 地上盤へ 安全ドアSW
151   LD      M1103  ; AGV光転送2or6 停止中 OUT2_X0C7
      AND     M1106  ; AGV光転送2or6 対向中OUT5_X0CA
      OUT     Y1017  ; 地上盤へ 搬入 AGV在席
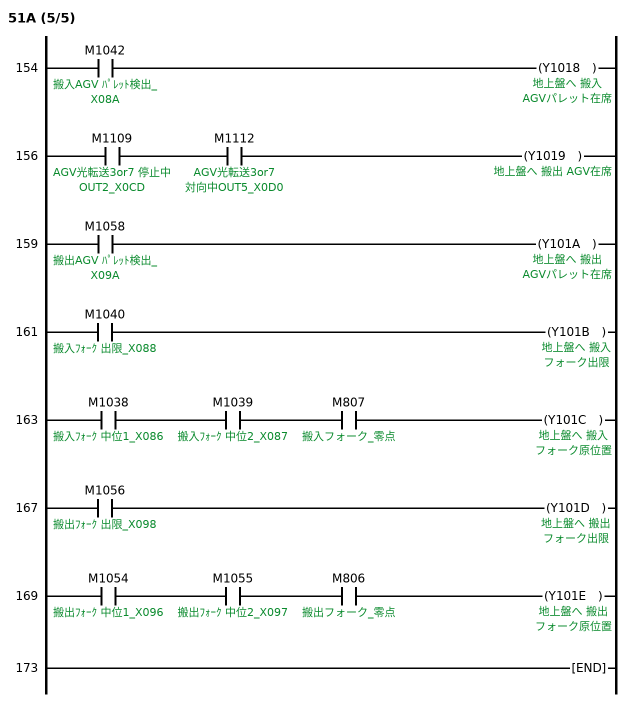
154   LD      M1042  ; 搬入AGV ﾊﾟﾚｯﾄ検出_X08A
      OUT     Y1018  ; 地上盤へ 搬入 AGVパレット在席
156   LD      M1109  ; AGV光転送3or7 停止中 OUT2_X0CD
      AND     M1112  ; AGV光転送3or7 対向中OUT5_X0D0
      OUT     Y1019  ; 地上盤へ 搬出 AGV在席
159   LD      M1058  ; 搬出AGV ﾊﾟﾚｯﾄ検出_X09A
      OUT     Y101A  ; 地上盤へ 搬出 AGVパレット在席
161   LD      M1040  ; 搬入ﾌｫｰｸ 出限_X088
      OUT     Y101B  ; 地上盤へ 搬入 フォーク出限
163   LD      M1038  ; 搬入ﾌｫｰｸ 中位1_X086
      AND     M1039  ; 搬入ﾌｫｰｸ 中位2_X087
      AND     M807  ; 搬入フォーク_零点
      OUT     Y101C  ; 地上盤へ 搬入 フォーク原位置
167   LD      M1056  ; 搬出ﾌｫｰｸ 出限_X098
      OUT     Y101D  ; 地上盤へ 搬出 フォーク出限
169   LD      M1054  ; 搬出ﾌｫｰｸ 中位1_X096
      AND     M1055  ; 搬出ﾌｫｰｸ 中位2_X097
      AND     M806  ; 搬出フォーク_零点
      OUT     Y101E  ; 地上盤へ 搬出 フォーク原位置
173   END
END_PROGRAM

// device comments not shown above
X20  ; ユニットREADY
X21  ; 基本パラメータ登録正常完了
X22  ; 基本パラメータ登録異常完了
X23  ; 基本パラメータ登録有無
X24  ; 自動交信パラメータ登録正常完了
X25  ; 自動交信パラメータ登録異常完了
X26  ; 自動交信機能動作状態
X27  ; 自動交信機能異常状態
X28  ; MODBUSﾃﾞﾊﾞｲｽ割付ﾊﾟﾗﾒｰﾀ登録正常
X29  ; MODBUSﾃﾞﾊﾞｲｽ割付ﾊﾟﾗﾒｰﾀ登録異常
X2A  ; MODBUSﾃﾞﾊﾞｲｽ割付ﾊﾟﾗﾒｰﾀ登録有無
X3B  ; COM.ERR.LED点灯状態
X3C  ; PINGテスト完了
X3F  ; ウォッチドグタイマエラー
X41  ; 基本パラメータ登録正常完了
X42  ; 基本パラメータ登録異常完了
X44  ; 自動交信パラメータ登録正常完了
X45  ; 自動交信パラメータ登録異常完了
X46  ; 自動交信機能動作状態
X47  ; 自動交信機能異常状態
X48  ; MODBUSﾃﾞﾊﾞｲｽ割付ﾊﾟﾗﾒｰﾀ登録正常
X49  ; MODBUSﾃﾞﾊﾞｲｽ割付ﾊﾟﾗﾒｰﾀ登録異常
X4A  ; MODBUSﾃﾞﾊﾞｲｽ割付ﾊﾟﾗﾒｰﾀ登録有無
X5B  ; COM.ERR.LED点灯状態
X5C  ; PINGテスト完了
X5F  ; ウォッチドグタイマエラー
Y21  ; 基本パラメータ登録要求
Y24  ; 自動交信 ﾊﾟﾗﾒｰﾀ登録/起動要求
Y26  ; 自動交信機能停止要求
Y28  ; MODBUSﾃﾞﾊﾞｲｽ割付ﾊﾟﾗﾒｰﾀ登録要求
Y3B  ; COM.ERR.LED消灯要求
Y3C  ; PINGテスト実行要求
Y41  ; 基本パラメータ登録要求
Y44  ; 自動交信 ﾊﾟﾗﾒｰﾀ登録/起動要求
Y46  ; 自動交信機能停止要求
Y48  ; MODBUSﾃﾞﾊﾞｲｽ割付ﾊﾟﾗﾒｰﾀ登録要求
Y5B  ; COM.ERR.LED消灯要求
Y5C  ; PINGテスト実行要求
D2  ; GOTｵｰﾊﾞﾗｯﾌﾟｳｨﾝﾄﾞｳ2
D3  ; GOTｵｰﾊﾞﾗｯﾌﾟｳｨﾝﾄﾞｳ3
D4  ; GOTｵｰﾊﾞﾗｯﾌﾟｳｨﾝﾄﾞｳ4
D5  ; GOTｵｰﾊﾞﾗｯﾌﾟｳｨﾝﾄﾞｳ5
D10  ; GOTｼｽﾃﾑ信号1-1
D11  ; GOTｼｽﾃﾑ信号2-1
D13  ; 表示中ｳｨﾝﾄﾞｳ画面1番号
D14  ; 表示中ｳｨﾝﾄﾞｳ画面2番号
D15  ; 表示中ｳｨﾝﾄﾞｳ画面3番号
D16  ; 表示中ｳｨﾝﾄﾞｳ画面4番号
D17  ; 表示中ｳｨﾝﾄﾞｳ画面5番号
D107  ; 搬入ﾌｫｰｸ 現在値32ﾋﾞｯﾄ
D117  ; 搬出ﾌｫｰｸ 現在値32ﾋﾞｯﾄ
D314  ; 搬入 RFID読値 2
D315  ; 搬入 RFID読値 3
D316  ; 搬入 RFID読値 4
D317  ; 搬入 RFID読値 5
D318  ; 搬入 RFID読値 6
D321  ; 搬出 RFID読値 2
D322  ; 搬出 RFID読値 3
D323  ; 搬出 RFID読値 4
D324  ; 搬出 RFID読値 5
D325  ; 搬出 RFID読値 6
D601  ; 搬入 RFID読値 2
D602  ; 搬入 RFID読値 3
D603  ; 搬入 RFID読値 4
D604  ; 搬入 RFID読値 5
D605  ; 搬入 RFID読値 6
D611  ; 搬入台 RFID ﾄﾗｯｷﾝｸﾞ 2
D612  ; 搬入台 RFID ﾄﾗｯｷﾝｸﾞ 3
D613  ; 搬入台 RFID ﾄﾗｯｷﾝｸﾞ 4
D614  ; 搬入台 RFID ﾄﾗｯｷﾝｸﾞ 5
D615  ; 搬入台 RFID ﾄﾗｯｷﾝｸﾞ 6
D621  ; 搬出 RFID読値 2
D622  ; 搬出 RFID読値 3
D623  ; 搬出 RFID読値 4
D624  ; 搬出 RFID読値 5
D625  ; 搬出 RFID読値 6
D631  ; 搬出 ﾌｫｰｸ RFID トラキング 2
D632  ; 搬出 ﾌｫｰｸ RFID トラキング 3
D633  ; 搬出 ﾌｫｰｸ RFID トラキング 4
D634  ; 搬出 ﾌｫｰｸ RFID トラキング 5
D635  ; 搬出 ﾌｫｰｸ RFID トラキング 6
D1101  ; 搬出 フォーク部タスクID
D1102  ; 搬出 搬出台タスクID
D1103  ; 搬出 搬出台タスクID
D1403  ; 地上盤から STK搬入完了
D1409  ; 地上盤から STK搬出完了
D3029  ; 地上盤へ AGV搬出完了
D3103  ; 地上盤から STK搬入完了
D3109  ; 地上盤から STK搬出完了
M243  ; 搬入ﾌｫｰｸﾌﾞﾚｰｷ解除
M263  ; 搬出ﾌｫｰｸﾌﾞﾚｰｷ解除
M600  ; 搬入フォーク部在席
M605  ; 搬入AGV停止
M606  ; 搬入AGV準備
M607  ; 搬入AGVﾊﾟﾚｯﾄ在席
M626  ; 搬入台 STK搬入完了
M651  ; 搬出CV 減速位置
M655  ; 搬出AGV停止
M656  ; 搬出AGV準備
M657  ; 搬出AGVﾊﾟﾚｯﾄ在席
M670  ; 搬出AGV通過許可
M671  ; 搬出AGVl離れ中
M672  ; 搬出AGV本体検知
M675  ; 搬出準備完了
M678  ; 搬出台 STK搬出完了
M800  ; スタッカー搬出中
M801  ; スタッカー搬入中
M802  ; アラーム立ち上がり
M803  ; イニシャライズ完成
M804  ; イニシャライズ開始
M805  ; 起動立ち上がり
M808  ; 設備静止中
M809  ; Deliver_In.AGV通過許可
M810  ; Deliver_In.AGV本体検知
M811  ; Deliver_In.AGV進入中
M812  ; E_Stop
M1500  ; 電源 入_地上盤ﾖﾘ
M1501  ; 運転準備 入_地上盤ﾖﾘ
M1502  ; 重故障_地上盤ﾖﾘ
M1503  ; 軽故障_地上盤ﾖﾘ
M1504  ; 非常停止 正常_地上盤ﾖﾘ
M1510  ; 自動運転中_地上盤ﾖﾘ
M1511  ; ｻｲｸﾙ停止中_地上盤ﾖﾘ
M1512  ; 手動操作中_地上盤ﾖﾘ
M1513  ; 特殊操作中_地上盤ﾖﾘ
M1516  ; 自動ﾓｰﾄﾞ選択_地上盤ﾖﾘ
M1517  ; 手動ﾓｰﾄﾞ選択_地上盤ﾖﾘ
M1518  ; 連動ﾓｰﾄﾞ選択_地上盤ﾖﾘ
M1519  ; 単独ﾓｰﾄﾞ選択_地上盤ﾖﾘ
M1520  ; 管理者ﾓｰﾄﾞ選択_地上盤ﾖﾘ
M1542  ; 搬入RFID 再取得_地上盤ﾖﾘ
M1543  ; 搬出RFID 再取得_地上盤ﾖﾘ
M2003  ; 搬入側RFID手動書込み完了
M2004  ; 搬出側RFID手動書込み完了
M2999  ; 常時ON SD変更
T35  ; 搬入CV停止遅延
T45  ; 搬出CV停止遅延
T48  ; 搬出ﾌｫｰｸ定位置到着確認
T180  ; 搬入 RFID 不一致 遅延
T181  ; 搬出 計画未達 遅延
T182  ; 搬入 RFID 読取NG 遅延
T183  ; 搬出 RFID 読取NG 遅延
B0  ; 電源 入_地上盤ﾖﾘ
B1  ; 運転準備 入_地上盤ﾖﾘ
B2  ; 重故障_地上盤ﾖﾘ
B3  ; 軽故障_地上盤ﾖﾘ
B4  ; 非常停止 正常_地上盤ﾖﾘ
B0A  ; 自動運転中_地上盤ﾖﾘ
B0B  ; ｻｲｸﾙ停止中_地上盤ﾖﾘ
B0C  ; 手動操作中_地上盤ﾖﾘ
B0D  ; 特殊操作中_地上盤ﾖﾘ
B10  ; 自動ﾓｰﾄﾞ選択_地上盤ﾖﾘ
B11  ; 手動ﾓｰﾄﾞ選択_地上盤ﾖﾘ
B12  ; 連動ﾓｰﾄﾞ選択_地上盤ﾖﾘ
B13  ; 単独ﾓｰﾄﾞ選択_地上盤ﾖﾘ
B14  ; 管理者ﾓｰﾄﾞ選択_地上盤ﾖﾘ
B1A  ; 連動 起動_地上盤ﾖﾘ
B1B  ; 連動 ｻｲｸﾙ停止_地上盤ﾖﾘ
B20  ; STK搬入中_地上盤ﾖﾘ
B21  ; STK搬入完了_地上盤ﾖﾘ
B22  ; STK搬出中_地上盤ﾖﾘ
B23  ; STK搬出完了 _地上盤ﾖﾘ
B2A  ; 搬入 RFID 再取得_地上盤ﾖﾘ
B2B  ; 搬出 RFID 再取得_地上盤ﾖﾘ
B1000  ; 電源 入_地上盤ﾍ
B1001  ; 運転準備 入_地上盤ﾍ
B1002  ; 重故障_地上盤ﾍ
B1003  ; 軽故障_地上盤ﾍ
B1004  ; 非常停止 正常_地上盤ﾍ
B1005  ; 安全ﾄﾞｱｽｲｯﾁ正常_地上盤ﾍ
B1006  ; ﾗｲﾄｶｰﾃﾝ正常(CV側)_地上盤ﾍ
B1007  ; ﾗｲﾄｶｰﾃﾝ正常(AGV側)_地上盤ﾍ
B100A  ; 自動運転中_地上盤ﾍ
B100B  ; ｻｲｸﾙ停止中_地上盤ﾍ
B100C  ; 手動操作中_地上盤ﾍ
B100D  ; 特殊操作中_地上盤ﾍ
B1010  ; 自動ﾓｰﾄﾞ選択_地上盤ﾍ
B1011  ; 手動ﾓｰﾄﾞ選択_地上盤ﾍ
B1012  ; 連動ﾓｰﾄﾞ選択_地上盤ﾍ
B1013  ; 単独ﾓｰﾄﾞ選択_地上盤ﾍ
B1014  ; 管理者ﾓｰﾄﾞ選択_地上盤ﾍ
B1020  ; 搬入RFID 読取完了_地上盤ﾍ
B1021  ; 搬入RFID 読取 NG_地上盤ﾍ
B1022  ; 搬出RFID 読取完了_地上盤ﾍ
B1023  ; 搬出RFID 読取 NG_地上盤ﾍ
B1028  ; ﾗｲﾄｶｰﾃﾝ 1or7 無効_地上盤ﾍ
B1029  ; ﾗｲﾄｶｰﾃﾝ 2 無効_地上盤ﾍ
B102A  ; ﾗｲﾄｶｰﾃﾝ 3or5 無効_地上盤ﾍ
B102B  ; ﾗｲﾄｶｰﾃﾝ 4or6 無効_地上盤ﾍ
B1030  ; ｽﾀｯｶｰｸﾚｰﾝ 搬入 可_地上盤ﾍ
B1031  ; AGV 発進可_地上盤ﾍ
B1033  ; 搬入ｺﾝﾍﾞｱ動作中_地上盤ﾍ
B1034  ; 搬入ﾌｫｰｸ 動作中_地上盤ﾍ
B1035  ; 搬入ﾌｫｰｸﾘﾌﾄ 動作中_地上盤ﾍ
B1036  ; 搬入台ﾘﾌﾄ 動作中_地上盤ﾍ
B1037  ; 搬入AGV 在席_地上盤ﾍ
B1038  ; 搬入CV ﾊﾟﾚｯﾄ 在席_地上盤ﾍ
B1039  ; 搬入台ﾊﾟﾚｯﾄ 在席_地上盤ﾍ
B103A  ; 搬入ﾌｫｰｸ 零点_地上盤ﾍ
B103B  ; 搬入ﾌｫｰｸ 出限_地上盤ﾍ
B103C  ; 搬入ﾌｫｰｸﾘﾌﾀ 下降端_地上盤ﾍ
B103D  ; 搬入ﾌｫｰｸﾘﾌﾀ  上昇端_地上盤ﾍ
B103E  ; 搬入台ﾘﾌﾀ 下降端_地上盤ﾍ
B103F  ; 1搬入台ﾘﾌﾀ 上昇端_地上盤ﾍ
B1040  ; ｽﾀｯｶｰｸﾚｰﾝ搬出 可_地上盤ﾍ
B1041  ; 搬出AGV 発進可_地上盤ﾍ
B1043  ; 搬出ｺﾝﾍﾞｱ動作中_地上盤ﾍ
B1044  ; 搬出ﾌｫｰｸ 動作中_地上盤ﾍ
B1045  ; 搬出ﾌｫｰｸﾘﾌﾀ 動作中_地上盤ﾍ
B1046  ; 搬出台ﾘﾌﾀ 動作中_地上盤ﾍ
B1047  ; 搬出AGV 在席_地上盤ﾍ
B1048  ; 搬出フォーク部 在席_地上盤ﾍ
B1049  ; 搬出台ﾊﾟﾚｯﾄ 在席_地上盤ﾍ
B104A  ; 搬出ﾌｫｰｸ 零点_地上盤ﾍ
B104B  ; 搬出ﾌｫｰｸ 出限_地上盤ﾍ
B104C  ; 搬出ﾌｫｰｸﾘﾌﾀ 下降端_地上盤ﾍ
B104D  ; 搬出ﾌｫｰｸﾘﾌﾀ 上昇端_地上盤ﾍ
B104E  ; 搬出台ﾘﾌﾀ 下降端_地上盤ﾍ
B104F  ; 搬出台ﾘﾌﾀ 下降端_地上盤ﾍ
W1000  ; 搬入 RFID 読値
W1008  ; 搬入ST RFID ﾄﾗｯｷﾝｸﾞ
W1010  ; 搬出 RFID 読値
W1018  ; 搬出 ﾌｫｰｸ RFID トラキング
D3005.0  ; 地上盤へ 搬入AGV搬入完了
